# EPICS substitutions: evrSupport/Db/ioc/trigXL05.substitutions
# Trigger records
#
# refer to Sharepoint document: Controls | Timing | timingTriggers.xls
#
# Must also have pattern records
# Note: WID, DES, TEC are in terms of nSec and are unique per device
#
file evrDevTrig.db {
#      Device	      , Description   , EVR  ,  width ,desired  , EC delay   , EVR  , EVR,  IOC          , slope
#			                            Trigger       wrt TREF   wrt fiducial loca   unit                 1/119Mhz
  pattern { DEV       ,  DESC         , T    ,  WID   , DES     , TEC        , LOCA , UNIT, IOC          , ESLO
                      ,  PREC         , EGU  ,  DRVL  , DRVH    , EVG}
	{ TRIG:XL05:1: ,  "trigger 0"     , 0    ,  100   , 10      , LCLSBEAM   , XL05 , EV01, IOC:XL05:EV01, 8.40336692324359
                      ,  1            ,"nSec", -2.8E06, 2.8E06  , IN20:EV01}
	{ TRIG:XL05:2: ,  "trigger 1"     , 1    ,  100   , 10      , TS1_120_,  , XL05 , EV01, IOC:XL05:EV01, 8.40336692324359
                      ,  1            ,"nSec", -2.8E06, 2.8E06  , IN20:EV01}
	{ TRIG:XL05:3: ,  "trigger 2"     , 2    ,  100   , 10      , TS1_60_    , XL05 , EV01, IOC:XL05:EV01, 8.40336692324359
                      ,  1            ,"nSec", -2.8E06, 2.8E06  , IN20:EV01 }
	{ TRIG:XL05:4: ,  "trigger 3"     , 3    ,  100   , 10      , TS1_30_    , XL05 , EV01, IOC:XL05:EV01, 8.40336692324359
                      ,  1            ,"nSec", -2.8E06, 2.8E06  , IN20:EV01 }
	{ TRIG:XL05:5: ,  "trigger 4"     , 4    ,  100   , 10      , TS1_10_    , XL05 , EV01, IOC:XL05:EV01, 8.40336692324359
                      ,  1            ,"nSec", -2.8E06, 2.8E06  , IN20:EV01 }
	{ TRIG:XL05:6: ,  "trigger 5"     , 5    ,  100   , 10      , TS1_5_     , XL05 , EV01, IOC:XL05:EV01, 8.40336692324359
                      ,  1            ,"nSec", -2.8E06, 2.8E06  , IN20:EV01 }
	{ TRIG:XL05:7: ,  "trigger 6"     , 6    ,  100   , 10      , TS4_120_   , XL05 , EV01, IOC:XL05:EV01, 8.40336692324359
                      ,  1            ,"nSec", -2.8E06, 2.8E06  , IN20:EV01 }
	{ TRIG:XL05:8: ,  "trigger 7"     , 7    ,  100   , 10      , TS4_60_    , XL05 , EV01, IOC:XL05:EV01, 8.40336692324359
                      ,  1            ,"nSec", -2.8E06, 2.8E06  , IN20:EV01}
	{ TRIG:XL05:9: ,  "trigger 8"     , 8    ,  100   , 10      , TS4_30_    , XL05 , EV01, IOC:XL05:EV01, 8.40336692324359
                      ,  1            ,"nSec", -2.8E06, 2.8E06  , IN20:EV01 }
	{ TRIG:XL05:10:,  "trigger 9 "    , 9    ,  100   , 10      , TS4_10_    , XL05 , EV01, IOC:XL05:EV01, 8.40336692324359
                      ,  1            ,"nSec", -2.8E06, 2.8E06  , IN20:EV01 }
	{ TRIG:XL05:11:,  "trigger 10"    , A    ,  100   , 10      , TS4_5_     , XL05 , EV01, IOC:XL05:EV01, 8.40336692324359
                      ,  1            ,"nSec", -2.8E06, 2.8E06  , IN20:EV01}
	{ TRIG:XL05:12:,  "trigger 11"    , B    ,  100   , 10      , TS4_1_     , XL05 , EV01, IOC:XL05:EV01, 8.40336692324359
                      ,  1            ,"nSec", -2.8E06, 2.8E06  , IN20:EV01 }
	{ TRIG:XL05:13:,  "trigger 12"    , C    ,  100   , 10      , TS4_HALF_  , XL05 , EV01, IOC:XL05:EV01, 8.40336692324359
                      ,  1            ,"nSec", -2.8E06, 2.8E06  , IN20:EV01 }

}
